{attribute addProperty BoxType "EM7004-0000-0016"}
{attribute addProperty Id "DI_InputsAT %I*DI_Inputs_42B6F5B2128160ENC_Inputs_ChannelAT %I*ARRAY[0..3] OF ENC_Inputs_Channel_8F9896EF352440PLS_InputsAT %I*PLS_Inputs_213E75F71620DO_OutputsAT %Q*DO_Outputs_BF554446128160AO_Outputs_ChannelAT %Q*ARRAY[0..3] OF AO_Outputs_Channel_F57FA4F96480ENC_Outputs_ChannelAT %Q*ARRAY[0..3] OF ENC_Outputs_Channel_14754A39160200PLS_OutputsAT %Q*PLS_Outputs_F618EC1A810WcStateAT %I*WcState_F855686C1620InfoDataAT %I*InfoData_BC63D37F80100"}
{attribute addProperty CRC "1305365264"}
{attribute addProperty SizeInBites "952"}
{attribute addProperty SizeInBytes "119"}
TYPE EM7004_A38AEEB0 :
STRUCT
	{attribute addProperty Name "DI_Inputs"}
	DI_Inputs : DI_Inputs_42B6F5B2;
	{attribute addProperty Name "ENC_Inputs_Channel"}
	ENC_Inputs_Channel : ARRAY[0..3] OF ENC_Inputs_Channel_8F9896EF;
	{attribute addProperty Name "PLS_Inputs"}
	PLS_Inputs : PLS_Inputs_213E75F7;
	{attribute addProperty Name "DO_Outputs"}
	DO_Outputs : DO_Outputs_BF554446;
	{attribute addProperty Name "AO_Outputs_Channel"}
	AO_Outputs_Channel : ARRAY[0..3] OF AO_Outputs_Channel_F57FA4F9;
	{attribute addProperty Name "ENC_Outputs_Channel"}
	ENC_Outputs_Channel : ARRAY[0..3] OF ENC_Outputs_Channel_14754A39;
	{attribute addProperty Name "PLS_Outputs"}
	PLS_Outputs : PLS_Outputs_F618EC1A;
	{attribute addProperty Name "WcState"}
	WcState : WcState_F855686C;
	{attribute addProperty Name "InfoData"}
	InfoData : InfoData_BC63D37F;
END_STRUCT
END_TYPE

(* stored: Version 1.2.0.0, ProductVersion 3.1.4024.9
   DUT EM7004_A38AEEB0: Id {598cb1b6-3094-4e98-9f7d-d798d2ee64d6} *)
